// TwinCAT 3 PLC project StatePLC
// ProgramVersion: 3.1.4023.0
// libraries:
//   Tc2_Standard, * (Beckhoff Automation GmbH)
//   Tc2_System, * (Beckhoff Automation GmbH)
//   Tc3_Module, * (Beckhoff Automation GmbH)
// project tree:
//   DUTs/ E_STATES.TcDUT
//   / PlcTask.TcTTO
//   POUs/ AbstractState.TcPOU, I_State.TcIO, I_Statehandler.TcIO, LogString.TcPOU, MAIN.TcPOU, State1.TcPOU, State2.TcPOU, StateExample.TcPOU
// real-time tasks:
//   TASK PlcTask: cycle T#10ms, priority 20, ADS port 350

CONFIGURATION StatePLC
    RESOURCE PLC ON TwinCAT3
        TASK PlcTask(INTERVAL := T#10ms, PRIORITY := 20);
        PROGRAM MAIN WITH PlcTask : MAIN;
    END_RESOURCE
END_CONFIGURATION

// ---- DUTs/E_STATES.TcDUT
{attribute 'qualified_only'}
{attribute 'strict'}
TYPE E_STATES :
(
	eState1 := 0,
	eState2
);
END_TYPE

// ---- POUs/I_State.TcIO
INTERFACE I_State

METHOD PUBLIC Handle : BOOL
END_METHOD

END_INTERFACE

// ---- POUs/I_Statehandler.TcIO
INTERFACE I_Statehandler

METHOD SetState : BOOL
VAR_INPUT
	eNewState: E_STATES;
END_VAR
END_METHOD

END_INTERFACE

// ---- POUs/MAIN.TcPOU
PROGRAM MAIN
VAR
	fbStateExample: StateExample;
END_VAR

fbStateExample();

END_PROGRAM

// ---- POUs/StateExample.TcPOU
FUNCTION_BLOCK StateExample IMPLEMENTS I_Statehandler
VAR
	// Interface pointer to THIS statehandler
	ipSH: I_Statehandler := THIS^;
	
	// State FBs
	fbState1: State1(ipSH);
	fbState2: State2(ipSH);

	// Interface pointer to the current state
	ipState: I_State := fbState1;
END_VAR

IF ipState <> 0 THEN
	ipState.Handle();
END_IF

METHOD SetState : BOOL
VAR_INPUT
	eNewState	: E_STATES;
END_VAR
CASE eNewState OF
	E_STATES.eState1:
		ipState := fbState1;
		
	E_STATES.eState2:
		ipState := fbState2;

	ELSE
		ADSLOGSTR(msgCtrlMask := ADSLOG_MSGTYPE_ERROR, msgFmtStr := 'unknown state', strArg := '');

END_CASE
END_METHOD

END_FUNCTION_BLOCK

// ---- POUs/State1.TcPOU
FUNCTION_BLOCK State1 EXTENDS AbstractState

METHOD Handle : BOOL
fbTON(IN := TRUE, PT := T#7s);
IF fbTON.Q THEN
	LogString(sString := 'Timer in State 1 fired. Changing State to State 2.');
	ipStatehandler.SetState(eNewState := E_STATES.eState2);
	fbTON(IN := FALSE);
END_IF
END_METHOD

END_FUNCTION_BLOCK

// ---- POUs/AbstractState.TcPOU
FUNCTION_BLOCK ABSTRACT AbstractState IMPLEMENTS I_State
VAR_INPUT
	ipStatehandler: I_Statehandler;
END_VAR
VAR
	fbTON: TON;
END_VAR

METHOD FB_init : BOOL
VAR_INPUT
	bInitRetains : BOOL; // if TRUE, the retain variables are initialized (warm start / cold start)
	bInCopyCode : BOOL;  // if TRUE, the instance afterwards gets moved into the copy code (online change)
	ipStatehandler: I_Statehandler;
END_VAR
THIS^.ipStatehandler := ipStatehandler;
END_METHOD

METHOD ABSTRACT Handle : BOOL
END_METHOD

END_FUNCTION_BLOCK

// ---- POUs/LogString.TcPOU
FUNCTION LogString : BOOL
VAR_INPUT
	sString: T_MaxString;
END_VAR

ADSLOGSTR(
	msgCtrlMask := ADSLOG_MSGTYPE_HINT,
	msgFmtStr := '%s',
	strArg := sString
);

END_FUNCTION

// ---- POUs/State2.TcPOU
FUNCTION_BLOCK State2 EXTENDS AbstractState

METHOD Handle : BOOL
fbTON(IN := TRUE, PT := T#7s);
IF fbTON.Q THEN
	LogString(sString := 'Timer in State 2 fired. Changing State to State 1.');
	ipStatehandler.SetState(eNewState := E_STATES.eState1);
	fbTON(IN := FALSE);
END_IF
END_METHOD

END_FUNCTION_BLOCK
